(* PLC project Drehtisch, KW-Software MULTIPROG 5.35 *)
(* stored: companyURL www.kw-software.com, productRelease Build 434, creationDateTime 2012-11-08T15:33:09, version 1352385189, modificationDateTime 2012-11-08T15:33:09 *)

(* Layer 3: Ablaufebene (Version 2: 1 Sensor mittig) --> Greift auf Layer 2 zu. Der FB spiegelt die Funktion "Transport nach x, dreh" eines Werkstücks wider. Der Unterschied zum FB "Drehen" aus Layer 2 besteht darin, dass der Drehablauf neben dem reinen Drehen des Drehtisches auch die Übernahme/Übergabe und das Transportieren des Werkstücks umfasst. Die Ansteuerung der fünf Werkstückpositionszustände (0, 1, 2, 3 und aus) wird durch drei Positionsvariablen (Position1/2/3_WK) realisiert. Die Ansteuerung der fünf Transportzielzustände (0, 1, 2, 3 und aus) wird durch drei Positionsvariablen (Transportrichtung1/2/3) realisiert. Dabei sind die Positionen folgendermaßen verteilt: Wenn der Drehtisch ist in der Ausgangsposition befindet (waagerecht), dann ist: - 0 befindet sich links - 1 befindet sich oben - 2 befindet sich rechts - 3 befindet sich unten Im Anfangsschritt findet kein Drehablauuf statt - kein Drehen/Transportieren/Übergeben/Übernehmen (Motoren aus). Je nach Setzen der Inputvariablen (alternative Verzweigung) wird der Drehtisch nach links oder rechts gedreht, um das Werkstück an der richtigen Position übernehmen zu können (hierzu wird die Position1/2/3_WK ausgewertet) - die Transition "T_xxx_ein" schaltet. Es ist aber auch möglich, dass kein Positionieren des Tisches nötig ist, wenn er bereits in der korrekten Position steht. Damit wird ein Zustand eingenommen, der erstmal alle Motoren stoppt (Wichtig ist, dass der Drehmotor gestoppt wird.). Nach Auswertung der Bedingungen wird anschließend der Zustand eingenommen, in dem ein Werkstück von der entsprechenden Seite übernommen wird. Liefert FB "Übernahme_gabe" das Quittierungssignal, dass erfolgreich übernommen wurde, schaltet die Transition. Damit wird ein Zustand eingenommen, der erstmal alle Motoren stoppt (Wichtig ist, dass der Transportbandmotor gestoppt wird.). Nach Auswertung der Bedingungen bzgl. der Zielposition, wohin das Werkstück transportiert werden soll, wird der Zustand eingenommen, in dem der Drehtisch in die korrekte Position gedreht wird (falls nötig), um das Werkstück korrekt zu übergeben. Liefert FB "Drehen" das Quittierungssignal, dass erfolgreich gedreht wurde, schaltet die Transition. Damit wird ein Zustand eingenommen, der erstmal alle Motoren stoppt (Wichtig ist, dass der Drehmotor gestoppt wird.). Nach Auswertung der Bedingungen, ob das Werkstück überhaupt über den Drehtisch transportiert werden muss, wird der Zustand eingenommen, in dem der Drehtisch das Werkstück transportiert. Ein Transportieren ist z.B. nicht nötig, wenn ein Werkstück "über Eck" transpportiert werden soll. Dabei wird das Werkstück an einem Ende des Drehtisches übernommen, der Drehtisch dreht sich um -90° und das Werkstück wird am selbem Ende wird übergeben. Liefert FB "Transportieren" das Quittierungssignal, dass erfolgreich transportiert wurde (falls nötig), schaltet die Transition. Damit wird ein Zustand eingenommen, der erstmal alle Motoren stoppt (Wichtig ist, dass der Transportbandmotor gestoppt wird.). Nach Auswertung der Bedingungen, an welcher Seite das Werkstück übergeben werden muss, wird der Zustand eingenommen, in dem der Drehtisch das Werkstück übergibt. Wurde erfolgreich übergeben, so ist der Drehablauf abgeschlossen. Dabei wird auch eine Statusvariable gesetzt (GDx_xxx), die den erfolgreichen Drehablauf quittiert, sodass die übergeordnete Steuerung weiß, wann der Transportvorgang des Drehtisches abgeschlossen ist. FB-Schnittstellen: --------------- Eingangsvariablen: - Transportrichtung1 - Transportrichtung2 - Transportrichtung3 - Position1_WK - Position2_WK - Position3_WK Ausgangsvariablen: - GDx_links - GDx_rechts Auftretende Warnungen "Instanz 'FB_xxx' mehrfach verwendet!": Hier ein Textauszug aus der Multiprog-Hilfe: "Die Warnung kann auch in einem Code-Arbeitsblatt in AS auftreten, wenn Sie dieselbe Instanz in verschiedenen Aktionen verwendet haben. Wenn nur eine Instanz zu einem Zeitpunkt ausgeführt wird, ist die Warnung für Sie ohne Bedeutung." *)
FUNCTION_BLOCK Transport_zu_x_dreh
  VAR_INPUT
    Transportrichtung1 : BOOL := FALSE;  (* Inputvariable: Gibt an, wohin das Werkstück transportiert werden soll. *)
    Transportrichtung2 : BOOL := FALSE;  (* Inputvariable: Gibt an, wohin das Werkstück transportiert werden soll. *)
    Transportrichtung3 : BOOL := FALSE;  (* Inputvariable: Gibt an, wohin das Werkstück transportiert werden soll. *)
    Position1_WK : BOOL := FALSE;  (* Inputvariable: Gibt an, an welcher Position das Werkstück anliegt. *)
    Position2_WK : BOOL := FALSE;  (* Inputvariable: Gibt an, an welcher Position das Werkstück anliegt. *)
    Position3_WK : BOOL := FALSE;  (* Inputvariable: Gibt an, an welcher Position das Werkstück anliegt. *)
  END_VAR
  VAR
    FB_Uebernahme : Uebernahme_gabe;  (* Outputvariable vom FB "Uebernahme_gabe". Quittierungssignal für Übernahme *)
    FB_Uebergabe : Uebernahme_gabe;  (* Outputvariable vom FB "Uebernahme_gabe". Quittierungssignal für Übergabe *)
    Quittierungssignal_links1 : BOOL := FALSE;  (* Hilfsvariable: Hier wird der Output des Uebergabe/Transportieren-FBs eingetragen. Es wurde nach links übergeben. ODER es wurde nach links transportiert. *)
    Quittierungssignal_rechts1 : BOOL := FALSE;  (* Hilfsvariabel: Hier wird der Output des Uebergabe/Transportieren-FBs eingetragen. Es wurde nach rechts übergeben. ODER es wurde nach rechts transportiert. *)
  END_VAR
  VAR_OUTPUT
    GDx_links : BOOL := FALSE;  (* Quittierungssignal: Es wurde nach links transportiert. (GD = gedreht) *)
    GDx_rechts : BOOL := FALSE;  (* Quittierungssignal: Es wurde nach rechts transportiert. (GD = gedreht) *)
  END_VAR
  VAR
    Quittierungssignal_links2 : BOOL := FALSE;
    Quittierungssignal_rechts2 : BOOL := FALSE;
    Quittierungssignal_links3 : BOOL := FALSE;
    Quittierungssignal_rechts3 : BOOL := FALSE;
    Quittierungssignal_links4 : BOOL := FALSE;
    Quittierungssignal_rechts4 : BOOL := FALSE;
    Quittierungssignal_links5 : BOOL := FALSE;
    Quittierungssignal_rechts5 : BOOL := FALSE;
    FB_Drehen_pos : Drehen;  (* Outputvaribale vom FB "Drehen" *)
    FB_Drehen_dreh : Drehen;  (* Outputvariable vom FB "Drehen" *)
    Drehtisch_pos0 : BOOL := FALSE;  (* Hilfsvariable: Der Drehtisch befindet sich in der Aufgangsposition: Endlage 0. *)
    Drehtisch_pos1 : BOOL := FALSE;  (* Hilfsvariable: Der Drehtisch befidnet sich in Endlage 1. *)
    Drehtisch_dreh0 : BOOL := FALSE;  (* Hilfsvariable: Der Drehtisch befindet sich in der Aufgangsposition: Endlage 0. *)
    Drehtisch_dreh1 : BOOL := FALSE;  (* Hilfsvariable: Der Drehtisch befidnet sich in Endlage 1. *)
  END_VAR

(* transition T_Positionieren_l_ein *)
(*Auswertung der Startposition
...dann wird die Transition gesetzt und der Folgezustand wird eingenommen.*)

(*Der FB "Übernahme_gabe" aus Layer 2 wird jeweils für Linksbewegung instanziiert.*)
FB_Drehen_pos();

(*Der lokalen (Hilfs-)Variable "Quittierungssignal_links" wird der jeweilige Ausgangwert des FBs "Übernahme_gabe" zugewiesen.*)
Drehtisch_pos1 := FB_Drehen_pos.Endlage_1;

(*Wenn Werkstück an Position 0 anliegt und der Drehtisch sich in Endlage0 befindet oder
wenn das Werkstück an Position 2 anliegt und der Drehtisch sich in Endlage0 befindet.*)
IF Position1_WK = TRUE AND Position2_WK = TRUE AND Position3_WK = TRUE AND Drehtisch_pos1 = TRUE OR
Position1_WK = FALSE AND Position2_WK = TRUE AND Position3_WK = FALSE AND Drehtisch_pos1 = TRUE
	THEN T_Positionieren_l_ein := TRUE;
	ELSE T_Positionieren_l_ein := FALSE;
END_IF;
(* transition T_Positionieren_r_ein *)
(*Auswertung der Startposition
...dann wird die Transition gesetzt und der Folgezustand wird eingenommen.*)

(*Der FB "Übernahme_gabe" aus Layer 2 wird jeweils für Linksbewegung instanziiert.*)
FB_Drehen_pos();

(*Der lokalen (Hilfs-)Variable "Quittierungssignal_links" wird der jeweilige Ausgangwert des FBs "Übernahme_gabe" zugewiesen.*)
Drehtisch_pos0 := FB_Drehen_pos.Endlage_0;

(*Wenn Werkstück an Position 0 anliegt und der Drehtisch sich in Endlage0 befindet oder
wenn das Werkstück an Position 2 anliegt und der Drehtisch sich in Endlage0 befindet.*)
IF Position1_WK = TRUE AND Position2_WK = FALSE AND Position3_WK = FALSE AND Drehtisch_pos0 = TRUE OR
Position1_WK = FALSE AND Position2_WK = FALSE AND Position3_WK = TRUE AND Drehtisch_pos0 = TRUE
	THEN T_Positionieren_r_ein := TRUE;
	ELSE T_Positionieren_r_ein := FALSE;
END_IF;
(* transition T_Positionieren_l_aus *)
(*Statusvariablenabfrage Drehtisch positionieren zur Werkstückübernahme*)

(*Der FB "Übernahme_gabe" aus Layer 2 wird jeweils für Linksbewegung instanziiert.*)
FB_Drehen_pos();

(*Der lokalen (Hilfs-)Variable "Quittierungssignal_links" wird der jeweilige Ausgangwert des FBs "Übernahme_gabe" zugewiesen.*)
Quittierungssignal_links1 := FB_Drehen_pos.GD_0;

(*Wenn das Quittierungssignal TRUE ist, gilt das Werkstück als erfolgreich übernommen und die Transition wird gesetzt.*)
IF Quittierungssignal_links1 = TRUE 
	THEN T_Positionieren_l_aus := TRUE;
	ELSE T_Positionieren_l_aus := FALSE;
END_IF;
(* transition T_Positionieren_r_aus *)
(*Statusvariablenabfrage Drehtisch positionieren zur Werkstückübernahme*)

(*Der FB "Übernahme_gabe" aus Layer 2 wird jeweils für Linksbewegung instanziiert.*)
FB_Drehen_pos();

(*Der lokalen (Hilfs-)Variable "Quittierungssignal_links" wird der jeweilige Ausgangwert des FBs "Übernahme_gabe" zugewiesen.*)
Quittierungssignal_rechts1 := FB_Drehen_pos.GD_1;

(*Wenn das Quittierungssignal TRUE ist, gilt das Werkstück als erfolgreich übernommen und die Transition wird gesetzt.*)
IF Quittierungssignal_rechts1 = TRUE 
	THEN T_Positionieren_r_aus := TRUE;
	ELSE T_Positionieren_r_aus := FALSE;
END_IF;
(* transition T_Uebernehmen_l_ein *)
(*Übernehmen
...dann wird die Transition gesetzt und der Folgezustand wird eingenommen.*)

(*Wenn Werkstück an Position 2 oder 3 abliegt, dann Motor links drehen, damit Werkstück übernommen wird.*)
IF Position1_WK = FALSE AND Position2_WK = TRUE AND Position3_WK = FALSE OR
Position1_WK = FALSE AND Position2_WK = FALSE AND Position3_WK = TRUE
	THEN T_Uebernehmen_l_ein := TRUE;
	ELSE T_Uebernehmen_l_ein := FALSE;
END_IF;
(* transition T_Uebernehmen_r_ein *)
(*Übernehmen
...dann wird die Transition gesetzt und der Folgezustand wird eingenommen.*)

(*Wenn Werkstück an Position 0 oder 1 abliegt, dann Motor rechts drehen, damit Werkstück übernommen wird.*)
IF Position1_WK = TRUE AND Position2_WK = TRUE AND Position3_WK = TRUE OR
Position1_WK = TRUE AND Position2_WK = FALSE AND Position3_WK = FALSE
	THEN T_Uebernehmen_r_ein := TRUE;
	ELSE T_Uebernehmen_r_ein := FALSE;
END_IF;
(* transition T_Uebernehmen_l_aus *)
(*Statusvariablenabfrage. Werkstück übernommen*)

(*Der FB "Übernahme_gabe" aus Layer 2 wird jeweils für Linksbewegung instanziiert.*)
FB_Uebernahme();

(*Der lokalen (Hilfs-)Variable "Quittierungssignal_links" wird der jeweilige Ausgangwert des FBs "Übernahme_gabe" zugewiesen.*)
Quittierungssignal_links2 := FB_Uebernahme.UeG_UeN_links;

(*Wenn das Quittierungssignal TRUE ist, gilt das Werkstück als erfolgreich übernommen und die Transition wird gesetzt.*)
IF Quittierungssignal_links2 = TRUE 
	THEN T_Uebernehmen_l_aus := TRUE;
	ELSE T_Uebernehmen_l_aus := FALSE;
END_IF;
(* transition T_Uebernehmen_r_aus *)
(*Statusvariablenabfrage. Werkstück übernommen*)

(*Der FB "Übernahme_gabe" aus Layer 2 wird jeweils für Rechtsbewegung instanziiert.*)
FB_Uebernahme();

(*Der lokalen (Hilfs-)Variable "Quittierungssignal_rechts" wird der jeweilige Ausgangwert des FBs "Übernahme_gabe" zugewiesen.*)
Quittierungssignal_rechts2 := FB_Uebernahme.UeG_UeN_rechts;

(*Wenn das Quittierungssignal TRUE ist, gilt das Werkstück als erfolgreich übernommen und die Transition wird gesetzt.*)
IF Quittierungssignal_rechts2 = TRUE
	THEN T_Uebernehmen_r_aus := TRUE;
	ELSE T_Uebernehmen_r_aus := FALSE;
END_IF;
(* transition T_Drehung_l_ein *)
(*Auswertung der Zielposition
...dann wird die Transition gesetzt und der Folgezustand wird eingenommen.*)

(*Der FB "Übernahme_gabe" aus Layer 2 wird jeweils für Linksbewegung instanziiert.*)
FB_Drehen_dreh();

(*Der lokalen (Hilfs-)Variable "Quittierungssignal_links" wird der jeweilige Ausgangwert des FBs "Übernahme_gabe" zugewiesen.*)
Drehtisch_dreh1 := FB_Drehen_dreh.Endlage_1;

(*Wenn Werkstück nach 0 oder 2 transportiert werden soll und Endlage 1 ausgelöst ist, dann drehe Motor links*)
IF Transportrichtung1 = TRUE AND Transportrichtung2 = TRUE AND Transportrichtung3 = TRUE AND Drehtisch_dreh1 = TRUE OR
Transportrichtung1 = FALSE AND Transportrichtung2 = TRUE AND Transportrichtung3 = FALSE AND Drehtisch_dreh1 = TRUE
	THEN T_Drehung_l_ein := TRUE;
	ELSE T_Drehung_l_ein := FALSE;
END_IF;
(* transition T_Drehung_r_ein *)
(*Auswertung der Zielposition
...dann wird die Transition gesetzt und der Folgezustand wird eingenommen.*)

(*Der FB "Übernahme_gabe" aus Layer 2 wird jeweils für Linksbewegung instanziiert.*)
FB_Drehen_dreh();

(*Der lokalen (Hilfs-)Variable "Quittierungssignal_links" wird der jeweilige Ausgangwert des FBs "Übernahme_gabe" zugewiesen.*)
Drehtisch_dreh0 := FB_Drehen_dreh.Endlage_0;

(*Wenn Werkstück nach 1 oder 3 transportiert werden soll und Endlage 0 ausgelöst ist, dann drehe Motor links*)
IF Transportrichtung1 = TRUE AND Transportrichtung2 = FALSE AND Transportrichtung3 = FALSE AND Drehtisch_dreh0 = TRUE OR
Transportrichtung1 = FALSE AND Transportrichtung2 = FALSE AND Transportrichtung3 = TRUE AND Drehtisch_dreh0 = TRUE
	THEN T_Drehung_r_ein := TRUE;
	ELSE T_Drehung_r_ein := FALSE;
END_IF;
(* transition T_Drehung_l_aus *)
(*Statusvariablenabfrage Drehtisch positionieren zur Werkstückübernahme*)

(*Der FB "Übernahme_gabe" aus Layer 2 wird jeweils für Linksbewegung instanziiert.*)
FB_Drehen_dreh();

(*Der lokalen (Hilfs-)Variable "Quittierungssignal_links" wird der jeweilige Ausgangwert des FBs "Übernahme_gabe" zugewiesen.*)
Quittierungssignal_links3 := FB_Drehen_dreh.GD_0;

(*Wenn das Quittierungssignal TRUE ist, gilt das Werkstück als erfolgreich übernommen und die Transition wird gesetzt.*)
IF Quittierungssignal_links3 = TRUE 
	THEN T_Drehung_l_aus := TRUE;
	ELSE T_Drehung_l_aus := FALSE;
END_IF;
(* transition T_Drehung_r_aus *)
(*Statusvariablenabfrage Drehtisch positionieren zur Werkstückübernahme*)

(*Der FB "Übernahme_gabe" aus Layer 2 wird jeweils für Linksbewegung instanziiert.*)
FB_Drehen_dreh();

(*Der lokalen (Hilfs-)Variable "Quittierungssignal_links" wird der jeweilige Ausgangwert des FBs "Übernahme_gabe" zugewiesen.*)
Quittierungssignal_rechts3 := FB_Drehen_dreh.GD_1;

(*Wenn das Quittierungssignal TRUE ist, gilt das Werkstück als erfolgreich übernommen und die Transition wird gesetzt.*)
IF Quittierungssignal_rechts3 = TRUE 
	THEN T_Drehung_r_aus := TRUE;
	ELSE T_Drehung_r_aus := FALSE;
END_IF;
(* transition T_Uebergeben_l_ein *)
(*Wird vom Anwender oder vom darüberliegenden Layer die Entscheidung getroffen, dass das Transportband nach links befördern soll, 
dann wird die Transition gesetzt und der Folgezustand wird eingenommen.*)

(*Es wird nach links übergeben, wenn das Trabsportziel 0 oder 1 ist*)
IF Transportrichtung1 = TRUE AND Transportrichtung2 = TRUE AND Transportrichtung3 = TRUE OR
Transportrichtung1 = TRUE AND Transportrichtung2 = FALSE AND Transportrichtung3 = FALSE
	THEN T_Uebergeben_l_ein := TRUE;
	ELSE T_Uebergeben_l_ein := FALSE;
END_IF;
(* transition T_Uebergeben_r_ein *)
(*Wird vom Anwender oder vom darüberliegenden Layer die Entscheidung getroffen, dass das Transportband nach links befördern soll, 
dann wird die Transition gesetzt und der Folgezustand wird eingenommen.*)

(*Es wird nach rechts übergeben, wenn das Trabsportziel 2 oder 3 ist*)
IF Transportrichtung1 = FALSE AND Transportrichtung2 = TRUE AND Transportrichtung3 = FALSE OR
Transportrichtung1 = FALSE AND Transportrichtung2 = FALSE AND Transportrichtung3 = TRUE
	THEN T_Uebergeben_r_ein := TRUE;
	ELSE T_Uebergeben_r_ein := FALSE;
END_IF;
(* transition T_Drehablauf_l_aus *)
(*Statusvariablenabfrage. Uebergeben*)

(*Der FB "Übernahme_gabe" aus Layer 2 wird jeweils für Linksbewegung instanziiert.*)
FB_Uebergabe();

(*Der lokalen (Hilfs-)Variable "Quittierungssignal_links" wird der jeweilige Ausgangwert des FBs "Übernahme_gabe" zugewiesen.*)
Quittierungssignal_links5 := FB_Uebergabe.UeG_UeN_links;

(*Wenn das Quittierungssignal TRUE ist, gilt das Werkstück als erfolgreich übergeben und die Transition wird gesetzt.*)
IF Quittierungssignal_links5 = TRUE
	THEN T_Drehablauf_l_aus := TRUE;
	ELSE T_Drehablauf_l_aus := FALSE;
END_IF;
(* transition T_Drehablauf_r_aus *)
(*Statusvariablenabfrage. Uebergeben*)

(*Der FB "Übernahme_gabe" aus Layer 2 wird jeweils für Rechtsbewegung instanziiert.*)
FB_Uebergabe();

(*Der lokalen (Hilfs-)Variable "Quittierungssignal_links" wird der jeweilige Ausgangwert des FBs "Übernahme_gabe" zugewiesen.*)
Quittierungssignal_rechts5 := FB_Uebergabe.UeG_UeN_rechts;

(*Wenn das Quittierungssignal TRUE ist, gilt das Werkstück als erfolgreich übergeben und die Transition wird gesetzt.*)
IF Quittierungssignal_rechts5 = TRUE 
	THEN T_Drehablauf_r_aus := TRUE;
	ELSE T_Drehablauf_r_aus := FALSE;
END_IF;
(* transition T_sofort_weiter7 *)
(*In dieser Transition steckt keine Bedingung. Die Transition wird sofort gesetzt und der Folgezustand wird eingenommen.*)
(* transition T_sofort_weiter8 *)
(*In dieser Transition steckt keine Bedingung. Die Transition wird sofort gesetzt und der Folgezustand wird eingenommen.*)
(* transition T_kein_Positionieren *)
(*Wird vom Anwender oder vom darüberliegenden Layer die Entscheidung getroffen, dass das Transportband nach links befördern soll, 
dann wird die Transition gesetzt und der Folgezustand wird eingenommen.*)

(*Auswertung der Startposition
...dann wird die Transition gesetzt und der Folgezustand wird eingenommen.*)

(*Der FB "Übernahme_gabe" aus Layer 2 wird jeweils für Linksbewegung instanziiert.*)
FB_Drehen_pos();

(*Der lokalen (Hilfs-)Variable "Quittierungssignal_links" wird der jeweilige Ausgangwert des FBs "Übernahme_gabe" zugewiesen.*)
Drehtisch_pos0 := FB_Drehen_pos.Endlage_0;
Drehtisch_pos1 := FB_Drehen_pos.Endlage_1;


(*Wenn Werkstück an 0 oder 2 anliegt und Endlage 0 ausgelöst ist.*)
(*Wenn Werkstück an 1 oder 3 anliegt und Endlage 1 ausgelöst ist.*)
(*DANN ist kein Positionieren des Drehtisches nötig.*)
IF (Position1_WK = TRUE AND Position2_WK = TRUE AND Position3_WK = TRUE AND Drehtisch_pos0 = TRUE OR
Position1_WK = FALSE AND Position2_WK = TRUE AND Position3_WK = FALSE AND Drehtisch_pos0 = TRUE) OR
(Position1_WK = TRUE AND Position2_WK = FALSE AND Position3_WK = FALSE AND Drehtisch_pos1 = TRUE OR
Position1_WK = FALSE AND Position2_WK = FALSE AND Position3_WK = TRUE AND Drehtisch_pos1 = TRUE)
	THEN T_kein_Positionieren := TRUE;
	ELSE T_kein_Positionieren := FALSE;
END_IF;
(* transition T_keine_Drehung *)
(*Wird vom Anwender oder vom darüberliegenden Layer die Entscheidung getroffen, dass das Transportband nach links befördern soll, 
dann wird die Transition gesetzt und der Folgezustand wird eingenommen.*)

(*Auswertung der Startposition
...dann wird die Transition gesetzt und der Folgezustand wird eingenommen.*)

(*Der FB "Übernahme_gabe" aus Layer 2 wird jeweils für Linksbewegung instanziiert.*)
FB_Drehen_dreh();

(*Der lokalen (Hilfs-)Variable "Quittierungssignal_links" wird der jeweilige Ausgangwert des FBs "Übernahme_gabe" zugewiesen.*)
Drehtisch_dreh0 := FB_Drehen_dreh.Endlage_0;
Drehtisch_dreh1 := FB_Drehen_dreh.Endlage_1;


(*Wenn Werkstück nach 0 oder 2 trabsportiert werden soll und Endlage 0 ausgelöst ist.*)
(*Wenn Werkstück nach 1 oder 3 transportiert werden soll und Endlage 1 ausgelöst ist.*)
(*DANN ist kein Positionieren des Drehtisches nötig.*)
IF (Transportrichtung1 = TRUE AND Transportrichtung2 = TRUE AND Transportrichtung3 = TRUE AND Drehtisch_dreh0 = TRUE OR
Transportrichtung1 = FALSE AND Transportrichtung2 = TRUE AND Transportrichtung3 = FALSE AND Drehtisch_dreh0 = TRUE) OR
(Transportrichtung1 = TRUE AND Transportrichtung2 = FALSE AND Transportrichtung3 = FALSE AND Drehtisch_dreh1 = TRUE OR
Transportrichtung1 = FALSE AND Transportrichtung2 = FALSE AND Transportrichtung3 = TRUE AND Drehtisch_dreh1 = TRUE)
	THEN T_keine_Drehung := TRUE;
	ELSE T_keine_Drehung := FALSE;
END_IF;
INITIAL_STEP Motor_aus:
END_STEP
TRANSITION FROM Motor_aus TO Drehmotor_links_pos
  := T_Positionieren_l_ein;
END_TRANSITION
TRANSITION FROM Motor_aus TO Drehmotor_rechts_pos
  := T_Positionieren_r_ein;
END_TRANSITION
TRANSITION FROM Motor_aus TO Drehmotor_aus
  := T_kein_Positionieren;
END_TRANSITION
STEP Drehmotor_links_pos:
END_STEP
TRANSITION FROM Drehmotor_links_pos TO Drehmotor_aus
  := T_Positionieren_l_aus;
END_TRANSITION
STEP Drehmotor_rechts_pos:
END_STEP
TRANSITION FROM Drehmotor_rechts_pos TO Drehmotor_aus
  := T_Positionieren_r_aus;
END_TRANSITION
STEP Drehmotor_aus:
END_STEP
TRANSITION FROM Drehmotor_aus TO Motor_links_UeN
  := T_Uebernehmen_l_ein;
END_TRANSITION
TRANSITION FROM Drehmotor_aus TO Motor_rechts_UeN
  := T_Uebernehmen_r_ein;
END_TRANSITION
STEP Motor_links_UeN:
END_STEP
TRANSITION FROM Motor_links_UeN TO Motor_aus2
  := T_Uebernehmen_l_aus;
END_TRANSITION
STEP Motor_rechts_UeN:
END_STEP
TRANSITION FROM Motor_rechts_UeN TO Motor_aus2
  := T_Uebernehmen_r_aus;
END_TRANSITION
STEP Motor_aus2:
END_STEP
TRANSITION FROM Motor_aus2 TO Drehmotor_links_dreh
  := T_Drehung_l_ein;
END_TRANSITION
TRANSITION FROM Motor_aus2 TO Drehmotor_rechts_dreh
  := T_Drehung_r_ein;
END_TRANSITION
TRANSITION FROM Motor_aus2 TO Drehmotor_aus2
  := T_keine_Drehung;
END_TRANSITION
STEP Drehmotor_links_dreh:
END_STEP
TRANSITION FROM Drehmotor_links_dreh TO Drehmotor_aus2
  := T_Drehung_l_aus;
END_TRANSITION
STEP Drehmotor_rechts_dreh:
END_STEP
TRANSITION FROM Drehmotor_rechts_dreh TO Drehmotor_aus2
  := T_Drehung_r_aus;
END_TRANSITION
STEP Drehmotor_aus2:
END_STEP
TRANSITION FROM Drehmotor_aus2 TO Motor_links_UeG
  := T_Uebergeben_l_ein;
END_TRANSITION
TRANSITION FROM Drehmotor_aus2 TO Motor_rechts_UeG
  := T_Uebergeben_r_ein;
END_TRANSITION
STEP Motor_links_UeG:
END_STEP
TRANSITION FROM Motor_links_UeG TO Quittierung_l
  := T_Drehablauf_l_aus;
END_TRANSITION
STEP Motor_rechts_UeG:
END_STEP
TRANSITION FROM Motor_rechts_UeG TO Quittierung_r
  := T_Drehablauf_r_aus;
END_TRANSITION
STEP Quittierung_l:
END_STEP
TRANSITION FROM Quittierung_l TO Endschritt_3  (* T_sofort_weiter7 *)
  := TRUE;
END_TRANSITION
STEP Quittierung_r:
END_STEP
TRANSITION FROM Quittierung_r TO Endschritt_3  (* T_sofort_weiter8 *)
  := TRUE;
END_TRANSITION
STEP Endschritt_3:
END_STEP

ACTION Drehablauf_aus:
(*In diesem Zustand befindet sich der Motor im unbestromten Zustand - Also kein Transportieren/Übergeben/Übernehmen/Drehen.
Layer 3 greift auch Layer 2 "Transportieren", "Übernahme_gabe" und "Drehen" zu und setzt die Eingangsvariablen dieser FBs entsprechend.*)
FB_Uebernahme(Uebergeben := FALSE, Uebernehmen := FALSE);
FB_Uebergabe(Uebergeben := FALSE, Uebernehmen := FALSE);

FB_Drehen_pos(Drehen_links := FALSE, Drehen_rechts := FALSE);
FB_Drehen_dreh(Drehen_links := FALSE, Drehen_rechts := FALSE);
END_ACTION

ACTION Positionieren_l:
(*In diesem Zustand befindet sich der Motor in der Linksdrehung - Werkstück wird transportiert.
Layer 3 greift auch Layer 2 "Transportieren" zu und setzt die Eingangsvariablen dieses FBs entsprechend.*)
FB_Drehen_pos(Drehen_links := TRUE, Drehen_rechts := FALSE);
END_ACTION

ACTION Positionieren_r:
(*In diesem Zustand befindet sich der Motor in der Linksdrehung - Werkstück wird transportiert.
Layer 3 greift auch Layer 2 "Transportieren" zu und setzt die Eingangsvariablen dieses FBs entsprechend.*)
FB_Drehen_pos(Drehen_links := FALSE, Drehen_rechts := TRUE);
END_ACTION

ACTION Positionieren_aus:
(*In diesem Zustand befindet sich der Motor im unbestromten Zustand - Also kein Transportieren/Übergeben/Übernehmen/Drehen.
Layer 3 greift auch Layer 2 "Transportieren", "Übernahme_gabe" und "Drehen" zu und setzt die Eingangsvariablen dieser FBs entsprechend.*)
FB_Uebernahme(Uebergeben := FALSE, Uebernehmen := FALSE);
FB_Uebergabe(Uebergeben := FALSE, Uebernehmen := FALSE);

FB_Drehen_pos(Drehen_links := FALSE, Drehen_rechts := FALSE);
FB_Drehen_dreh(Drehen_links := FALSE, Drehen_rechts := FALSE);
END_ACTION

ACTION Uebernehmen_l:
(*In diesem Zustand befindet sich der Motor in der Linksdrehung - Werkstück wird übernommen.
Layer 3 greift auch Layer 2 "Übernahme_gabe" zu und setzt die Eingangsvariablen dieses FBs entsprechend.*)

(*von rechts übernehmen*)
FB_Uebernahme(Richtung := TRUE, Uebernehmen := TRUE, Uebergeben := FALSE);
END_ACTION

ACTION Uebernehmen_r:
(*In diesem Zustand befindet sich der Motor in der Rechtsdrehung - Werkstück wird übernommen.
Layer 3 greift auch Layer 2 "Übernahme_gabe" zu und setzt die Eingangsvariablen dieses FBs entsprechend.*)

(*von links übernehmen*)
FB_Uebernahme(Richtung := FALSE, Uebernehmen := TRUE, Uebergeben := FALSE);
END_ACTION

ACTION Uebernehmen_aus:
(*In diesem Zustand befindet sich der Motor im unbestromten Zustand - Also kein Transportieren/Übergeben/Übernehmen/Drehen.
Layer 3 greift auch Layer 2 "Transportieren", "Übernahme_gabe" und "Drehen" zu und setzt die Eingangsvariablen dieser FBs entsprechend.*)
FB_Uebernahme(Uebergeben := FALSE, Uebernehmen := FALSE);
FB_Uebergabe(Uebergeben := FALSE, Uebernehmen := FALSE);

FB_Drehen_pos(Drehen_links := FALSE, Drehen_rechts := FALSE);
FB_Drehen_dreh(Drehen_links := FALSE, Drehen_rechts := FALSE);
END_ACTION

ACTION Drehen_l:
(*In diesem Zustand befindet sich der Motor in der Linksdrehung - Werkstück wird transportiert.
Layer 3 greift auch Layer 2 "Transportieren" zu und setzt die Eingangsvariablen dieses FBs entsprechend.*)
FB_Drehen_dreh(Drehen_links := TRUE, Drehen_rechts := FALSE);
END_ACTION

ACTION Drehen_r:
(*In diesem Zustand befindet sich der Motor in der Linksdrehung - Werkstück wird transportiert.
Layer 3 greift auch Layer 2 "Transportieren" zu und setzt die Eingangsvariablen dieses FBs entsprechend.*)
FB_Drehen_dreh(Drehen_links := FALSE, Drehen_rechts := TRUE);
END_ACTION

ACTION Drehung_aus:
(*In diesem Zustand befindet sich der Motor im unbestromten Zustand - Also kein Transportieren/Übergeben/Übernehmen/Drehen.
Layer 3 greift auch Layer 2 "Transportieren", "Übernahme_gabe" und "Drehen" zu und setzt die Eingangsvariablen dieser FBs entsprechend.*)
FB_Uebernahme(Uebergeben := FALSE, Uebernehmen := FALSE);
FB_Uebergabe(Uebergeben := FALSE, Uebernehmen := FALSE);

FB_Drehen_pos(Drehen_links := FALSE, Drehen_rechts := FALSE);
FB_Drehen_dreh(Drehen_links := FALSE, Drehen_rechts := FALSE);
END_ACTION

ACTION Uebergeben_l:
(*In diesem Zustand befindet sich der Motor in der Linksdrehung - Werkstück wird übergeben.
Layer 3 greift auch Layer 2 "Übernahme_gabe" zu und setzt die Eingangsvariablen dieses FBs entsprechend.*)

(*nach links übergeben*)
FB_Uebergabe(Richtung := FALSE, Uebernehmen := FALSE, Uebergeben := TRUE);
END_ACTION

ACTION Uebergeben_r:
(*In diesem Zustand befindet sich der Motor in der Rechtsdrehung - Werkstück wird übergeben.
Layer 3 greift auch Layer 2 "Übernahme_gabe" zu und setzt die Eingangsvariablen dieses FBs entsprechend.*)

(*nach rechts übergeben*)
FB_Uebergabe(Richtung := TRUE, Uebernehmen := FALSE, Uebergeben := TRUE);
END_ACTION

ACTION Quittierung_links4:
(*Statusvariable: Wird gesetzt, wenn bei Linksdrehung erfolgreich der Drehablauf erledigt wurde.
Diese Signal ist nötig für übergeordnete Steuerungen.*)
GDx_links := TRUE;
END_ACTION

ACTION Quittierung_rechts4:
(*Statusvariable: Wird gesetzt, wenn bei Rechtsdrehung erfolgreich der Drehablauf erledigt wurde.
Diese Signal ist nötig für übergeordnete Steuerungen.*)
GDx_rechts := TRUE;
END_ACTION

ACTION Endschritt_Drehablauf:
(*In diesem Zustand befindet sich der Motor im unbestromten Zustand - Also kein Transportieren/Übergeben/Übernehmen/Drehen.
Layer 3 greift auch Layer 2 "Transportieren", "Übernahme_gabe" und "Drehen" zu und setzt die Eingangsvariablen dieser FBs entsprechend.*)
FB_Uebernahme(Uebergeben := FALSE, Uebernehmen := FALSE);
FB_Uebergabe(Uebergeben := FALSE, Uebernehmen := FALSE);

FB_Drehen_pos(Drehen_links := FALSE, Drehen_rechts := FALSE);
FB_Drehen_dreh(Drehen_links := FALSE, Drehen_rechts := FALSE);
END_ACTION
END_FUNCTION_BLOCK
